// SIMATIC S7-200 project (STEP 7-Micro/WIN), CPU 221 REL 01.10

SYMBOL_TABLE USER1
s1               I0.0     // khoi dong
s2               I0.1     // dung
y                Q0.0     // dong co
s3               I0.2     // reset
END_SYMBOL_TABLE

ORGANIZATION_BLOCK MAIN:OB1
TITLE=PROGRAM COMMENTS
BEGIN
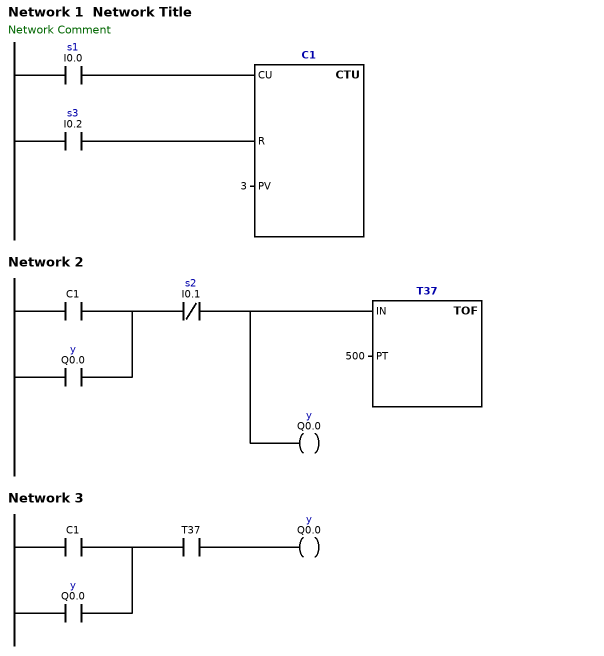
Network 1 // Network Title
// Network Comment
LD     s1:I0.0
LD     s3:I0.2
CTU    C1, 3
Network 2
LD     C1
O      y:Q0.0
AN     s2:I0.1
TOF    T37, 500
=      y:Q0.0
Network 3
LD     C1
O      y:Q0.0
A      T37
=      y:Q0.0
END_ORGANIZATION_BLOCK
